FUNCTION_BLOCK SimpleButton

VAR CONSTANT
	MAX_OUTPUTS_PER_LEVEL : INT := 3;
END_VAR

VAR_INPUT
	ID : INT;
	name : STRING := "Simple button";
	digitalInput : REFERENCE TO BOOL;
	outputs : REFERENCE TO ARRAY[1..MAX_OUTPUTS_PER_LEVEL] OF BOOL;
	runAsYouPress : BOOL := FALSE;
END_VAR
VAR_OUTPUT
END_VAR
VAR
	pressed : R_TRIG;
END_VAR

METHOD loop : BOOL
VAR_INPUT
END_VAR
pressed(CLK:= digitalInput);

IF runAsYouPress THEN
	setOutputs(state:= digitalInput);
ELSE
	IF pressed.Q THEN
		setOutputs(state:= TRUE);
	ELSE
		setOutputs(state:= FALSE);
	END_IF
END_IF
END_METHOD

METHOD setOutputs
VAR_INPUT
	state : BOOL;
END_VAR

VAR
	i : INT;
	state_as_text : STRING := 'abc';
END_VAR
state_as_text := TO_STRING(state);

GVL.EventLogger.print2(level:=TcEventSeverity.Info, str1:='set output to: %s', str2:= state_as_text);
FOR i := 1 TO MAX_OUTPUTS_PER_LEVEL BY 1 DO
	outputs[i] := state;
END_FOR
END_METHOD

END_FUNCTION_BLOCK

(* stored: Version 1.1.0.1, ProductVersion 3.1.4024.12
   POU SimpleButton: Id {8e1722dd-3bdd-4b96-a1d8-3587152ae0c6}, SpecialFunc None
   Method loop: Id {aa977121-eff7-4bf4-886a-ea3c6bcd0d1e}
   Method setOutputs: Id {b4040e0f-b48f-4a91-a4d6-98420882822c} *)
